# B&R Automation Studio project semesterProjekt_v002
Automation Studio 4.3.3.196

## Configuration Config1

### Task classes (Cpu.sw)
```
Cyclic#1 (cycle 1000 us, tolerance 1000 us):
  Program <- Program.prg
  reset <- reset.prg
Cyclic#4:
  emergencyS <- emergencyStop.prg
  TCP <- TCP.prg
VcDataObjects: Visu_R <- Visu_Resized.dob
Binaries: udbdef, TCData, vcrt, vcfntttf, Visu_R01, vcctext, Visu_R03, arial, vcmgr, vcpkat, vccovl, vccnum, vcpfar00, vcdsint, vcpfx20, vcpdvnc, vcshared, vcpdsw, vcfile, vcalarm, vccbtn, vcgclass, vcdsloc, arialbd, vcnet, vctcal, vcbclass, vccshape, Visu_R02, sysconf, Role, User, iomap, ashwd, asfw, arconfig, ashwac
Libraries: standard, astime, asieccon, fileio, dataobj, ashw, vcresman, AsMbTCP, runtime
```

### Hardware
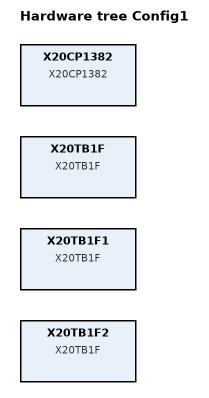
```
X20CP1382 : X20CP1382 v1.3.2.0  [X1 -> X1.SL; X2 -> X2.SL; X3 -> X3.SL]
  Module X1 (Type=X1, Virtual=true, Version=1.3.2.0)
    Connection (Connector=SS1, TargetModule=X20TB1F, TargetConnector=SS)
    Connection (Connector=SL, TargetModule=X20CP1382, TargetConnector=X1)
  Module X2 (Type=X2, Virtual=true, Version=1.3.2.0)
    Connection (Connector=SS1, TargetModule=X20TB1F1, TargetConnector=SS)
    Connection (Connector=SL, TargetModule=X20CP1382, TargetConnector=X2)
  Module X3 (Type=X3, Virtual=true, Version=1.3.2.0)
    Connection (Connector=SS1, TargetModule=X20TB1F2, TargetConnector=SS)
    Connection (Connector=SL, TargetModule=X20CP1382, TargetConnector=X3)
  Connector IF2:
    ActivateDevice = 1
    Mode = Manual
    InternetAddress = 192.168.0.103
    SubnetMask = 255.255.255.0
    Vnc1
    VncVcObjectName1 = Visu_R
    VncKeyMappingFile1 = VC\PS2-Keyboard.dis
    VncRefreshRate1 = 100
  ConfigurationID = semesterProjektTest_Config1
  VolatileGlobalPvSize = 655350
  SystemTick = 1000
  Cyclic1Duration = 1000
  Cyclic1Tolerance = 1000
X20TB1F : X20TB1F v1.0.0.0
X20TB1F1 : X20TB1F v1.0.0.0
X20TB1F2 : X20TB1F v1.0.0.0
```

## Logical view

Binary libraries used (declarations not repeated): operator, runtime, astime, AsIecCon, standard, AsMbTCP

### Global.var - Global variables
```iecst
VAR
	dirX : BOOL;
	dirY : BOOL;
	dirZ : BOOL;
	enabX : BOOL;
	enabY : BOOL;
	enabZ : BOOL;
	drawFunction : BOOL;
	input : ARRAY[0..1999999] OF UINT;
	posX : UDINT;
	posY : UDINT;
	posZ : UDINT;
	reset : BOOL;
	stepX : BOOL;
	stepY : BOOL;
	stepZ : BOOL;
	switch_X : BOOL;
	t : USINT;
	quit : BOOL;
	sharpen : UINT;
	status : USINT;
	testEnab : BOOL;
	z_move_down : BOOL;
	z_move_up : BOOL;
	y_move_right : BOOL;
	y_move_left : BOOL;
	x_move_right : BOOL;
	x_move_left : BOOL;
	sharpenderNeed : BOOL;
	switch_Z : BOOL;
	switch_Y : BOOL;
	percentage : REAL; (*%*)
	newLineX : UDINT;
	ValueZ : UINT;
	penLength : REAL;
	placeInString : UINT;
	placement : UINT;
	newLineHelper : UDINT;
END_VAR
```


### Program Logical/Program (IEC)

#### Main.st
```iecst
PROGRAM _INIT

	placeInString := 1;
	i := 0;
	sharpen := 1;
	activator := FALSE;
	testEnab:= FALSE;
	penLength := 0;
	sharpenderNeed:= 0;

END_PROGRAM

PROGRAM _CYCLIC
	ValueZ := REAL_TO_INT(penLength**1.5);

	IF (reset = FALSE AND testEnab = FALSE AND penLength > 5 ) THEN
//		percentage:= (UINT_TO_REAL(placeInString)/LEN(input))*100;

		IF (enabX = FALSE) THEN
			status:= 2;
		END_IF

		IF (i = 30) THEN
			placeInString := placeInString + 1;
			i := 0;
		END_IF
		placement := input[placeInString];

		// here the robot will move to the shapener, sharpen the pencil and move back to were it came from
		IF (sharpen = 1200 AND sharpenderNeed) THEN //!!!!!
			IF (posZ > 300 AND tempX > 0 AND activator = FALSE) THEN  // !!!!!!
				dirZ := TRUE;
				stepZ := NOT stepZ;
				IF (stepZ = FALSE) THEN
					posZ := posZ -1;
				END_IF

			ELSIF (tempX > 0 AND posZ = 300 AND activator = FALSE)THEN //!!!!!
				dirX := FALSE;
				stepX := NOT stepX;
				IF (stepX = FALSE) THEN
					tempX := tempX -1;
				END_IF

			ELSIF (tempX = 0 AND posZ < 1200 AND activator = FALSE) THEN //!!!!!
				dirZ := FALSE;
				stepZ := NOT stepZ;
				IF (stepZ = FALSE) THEN
					posZ := posZ +1;
				END_IF

			ELSIF (tempX = 0 AND posZ = 1200 AND activator = FALSE) THEN //!!!!!!
				timer.IN := TRUE;
				timer.PT := T#10000ms;
				IF timer.Q THEN
					activator := TRUE;
				END_IF

			ELSIF  (tempX = 0 AND posZ > 300 AND activator = TRUE) THEN//!!!!!
				dirZ := TRUE;
				stepZ := NOT stepZ;
				IF (stepZ = FALSE) THEN
					posZ := posZ - 1;
				END_IF

			ELSIF (tempX < posX  AND posZ = 300 AND activator = TRUE) THEN //!!!!!
				dirX := TRUE;
				stepX := NOT stepX;
				IF (stepX = FALSE) THEN
					tempX := tempX +1;
				END_IF

			ELSIF (tempX = posX  AND posZ = 300 AND activator = TRUE) THEN //!!!!!!
				sharpen := 0;
				activator := FALSE;

			END_IF

		ELSE
			// here the robot will draw
			IF (placement = 21041 AND i < 30) THEN
				IF (posZ < (3200-ValueZ)) THEN  // !!!!!!
						dirZ := TRUE;
						stepZ := NOT stepZ;
						IF (stepZ = FALSE) THEN
							posZ := posZ +1;
						END_IF

					ELSE
						dirX := TRUE;
						stepX := NOT stepX;
						IF (stepX = FALSE) THEN
							posX := posX + 1;
							newLineX := newLineX +1;
							sharpen := sharpen + 1;
							tempX := posX;
						END_IF
						i := i + 1;
					END_IF

			//dont draw
			ELSIF placement = 21040 AND i < 30) THEN

				IF (posZ > (2900-ValueZ)) THEN  // !!!!!!
						dirZ := FALSE;
						stepZ := NOT stepZ;
						IF (stepZ = FALSE) THEN
							posZ := posZ -1;
						END_IF

					ELSE
						dirX := TRUE;
						stepX := NOT stepX;
						IF (stepX = FALSE) THEN
							posX := posX +1;
							newLineX := newLineX +1;
						END_IF
						i := i + 1;

				ELSIF (i = 3) THEN
					placeInString := placeInString + 1;
					i := 0;

//				ELSE
//					placeInString := placeInString + 1;

				END_IF

//			ELSIF (placement = '1' OR placement = '0') THEN
//				placeInString := placeInString + 1;

			ELSIF (placement = 20016 OR placement = 20017) THEN
				IF (posZ > (2900-ValueZ) )THEN  // !!!!!!
					dirZ := FALSE;
					stepZ := NOT stepZ;
					IF (stepZ = FALSE) THEN
						posZ := posZ -1;
					END_IF
				ELSIF (posZ = (2900-ValueZ)) AND (newLineX >= (newLineHelper)) THEN//!!!!
					dirX := FALSE;
					stepX := NOT stepX;
					IF (stepX = FALSE) THEN
						posX := posX - 1;
						newLineX := newLineX -1;
					END_IF

				ELSIF ((posZ = (2900-ValueZ)) AND (newLineX <= newLineHelper) AND (i <= 30)(* OR ( posZ = 0)*)) THEN
					dirY := TRUE;
					stepY := NOT stepY;
					IF (stepY = FALSE) THEN
						posX := posX - 1;
						newLineX := newLineX -1;

					END_IF

					i := i +1;
				END_IF

				IF i = 20 THEN
					newLineHelper := newLineHelper - 12 ;

				END_IF

			ELSIF (placement = 20785 or placement = 20784) THEN

				quit := TRUE;
			END_IF

		END_IF

	END_IF
END_PROGRAM

PROGRAM _EXIT
	(* Insert code here *)

END_PROGRAM
```

### Program Logical/reset (IEC)

#### Main.st
```iecst
PROGRAM _INIT
	reset := TRUE;//!!!!!!!!
	resetX := 0;
	resetY := 0;
	resetZ := 0;

	quit := FALSE;
	status := 1;
	testEnab := TRUE;//!!!!!!
	posX := 0;
	posY := 0;
	posZ := 0;

END_PROGRAM

PROGRAM _CYCLIC

// resets x-, y- and z-axis.
	IF (reset = TRUE AND testEnab = FALSE) THEN
		IF switch_X = TRUE AND resetX = 0  THEN
			enabX:= FALSE;
			dirX:= FALSE;
			stepX := NOT stepX;
		ELSIF switch_X = FALSE THEN
			resetX := 1;
			dirX:= TRUE;
			stepX := NOT stepX;
		END_IF

		IF switch_Y = TRUE AND resetY = 0 THEN
			enabY:= FALSE;
			dirY:= FALSE;
			stepY := NOT stepY;
		ELSIF switch_Y = FALSE THEN
			resetY := 1;
			dirY:= TRUE;
			stepY := NOT stepY;
		END_IF

		IF switch_Z = TRUE AND resetZ = 0 THEN
			enabZ:= FALSE;
			dirZ:= FALSE;
			stepZ := NOT stepZ;
		ELSIF switch_Z = FALSE THEN
			resetZ := 1;
			dirZ:= TRUE;
			stepZ := NOT stepZ;
		END_IF
// sets the position of the variables posX, posY and posZ
		timer.IN := TRUE;
		timer.PT := T#100ms;
		IF timer.Q THEN
			IF resetX = 1 AND resetY = 1 AND resetZ = 1 THEN
				posX := 0;
				posY := 0;
				posZ := 0;
				resetX := 2;
			END_IF
			timer.IN := FALSE;
		END_IF

	// if start-button pressed, then go to start position
		IF quit = FALSE AND resetX = 2 THEN
			IF posX < 1900 THEN
				dirX := TRUE;
				stepX := NOT stepX;
				IF (stepX = FALSE) THEN
					posX := posX +1;
				END_IF
			ELSE
				reset:= FALSE;
				resetX := 0;
				resetY := 0;
				resetZ := 0;
				newLineX :=  2294967295;
				newLineHelper := 2294967295;
			END_IF
		END_IF
	END_IF

	// move x-axis left
	IF (x_move_left AND testEnab) THEN
		stepX := NOT stepX;
		dirX := TRUE;
		IF stepX = FALSE THEN
			posX := posX +1;
		END_IF
	END_IF

	// move x-axis right
	IF (x_move_right AND testEnab) THEN
		stepX := NOT stepX;
		dirX := FALSE;
		IF stepX = FALSE THEN
			posX := posX -1;
		END_IF
	END_IF

	// move y-axis left
	IF (y_move_left AND testEnab) THEN
		stepY := NOT stepY;
		dirY := TRUE;
		IF stepY = FALSE THEN
			posY := posY +1;
		END_IF
	END_IF

	// move y-axis right
	IF (y_move_right AND testEnab) THEN
		stepY := NOT stepY;
		dirY := FALSE;
		IF stepY = FALSE THEN
			posY := posY -1;
		END_IF
	END_IF

	// move z-axis up
	IF (z_move_up AND testEnab) THEN
		stepZ := NOT stepZ;
		dirZ := FALSE;
		IF stepZ = FALSE THEN
			posZ := posZ -1;
		END_IF
	END_IF

	// move z-axis down
	IF (z_move_down AND testEnab) THEN
		stepZ := NOT stepZ;
		dirZ := TRUE;
		IF stepZ = FALSE THEN
			posZ := posZ +1;
		END_IF
	END_IF

	timer();
END_PROGRAM

PROGRAM _EXIT
	(* Insert code here *)

END_PROGRAM
```

### Program Logical/emergencyStop (IEC)

#### Variables.var
```iecst
VAR
	emergencyStop : BOOL;
	reset_quit : BOOL;
END_VAR
```

#### Main.st
```iecst
PROGRAM _INIT
	(* Insert code here *)
	reset_quit := FALSE;
	emergencyStop := FALSE;

END_PROGRAM

PROGRAM _CYCLIC
	IF (emergencyStop) THEN
		enabX := TRUE;
		enabY := TRUE;
		enabZ := TRUE;
		status := 0;

	END_IF

	IF (reset_quit) THEN
		reset := TRUE;
		quit := TRUE;
		status := 1;
		reset_quit := FALSE;
		placeInString :=1;

	END_IF

END_PROGRAM

PROGRAM _EXIT
	(* Insert code here *)

END_PROGRAM
```

- Visualisation Logical/Visu_Resized (not shown)

### Program Logical/TCP (IEC)

#### Main.st
```iecst
PROGRAM _INIT
	state := 1;

END_PROGRAM

PROGRAM _CYCLIC
	CASE state OF
		1:
			tcp1.enable := TRUE;
			tcp1.port := 12345;
			tcp1.options := tcpOPT_REUSEADDR;
			tcp1();
			IF tcp1.status = 0 THEN
				state := 10;
			END_IF

		10:
			tcp2.enable := TRUE;
			tcp2.ident := tcp1.ident;
			tcp2();
			IF tcp2.status = 0 THEN
				state := 20;
			END_IF

		20:
			tcp3.enable := TRUE;
			tcp3.ident := tcp2.identclnt;
			tcp3.pData := ADR(reciveData);
			tcp3.datamax := SIZEOF (reciveData);
			tcp3();
			IF tcp3.status = 0 THEN
				sendData := reciveData;
				//				FOR i := 0 TO i = 2000 BY i + 1 DO
				//					test.IN := reciveData[i];
				//					input := CONCAT(input, test.Q);
				//				END_FOR
				state := 30;

			END_IF

		30:
			tcp4.enable := TRUE;
			tcp4.ident := tcp2.identclnt;
			tcp4.pData := ADR(sendData);
			tcp4.datalen := brsstrlen(ADR(sendData));
			tcp4();
			IF tcp4.status = 0 THEN
				state := 40;
			END_IF

		40:
			tcp5.enable := TRUE;
			tcp5.ident := tcp2.identclnt;
			tcp5();
			IF tcp5.status = 0 THEN
				tcp2.enable := FALSE;
				state := 10;

				//				FOR i := 0 TO i < 200 BY i + 1 DO
				//					reciveData[i] := 0;
				//				END_FOR
			END_IF
	END_CASE
	test();
END_PROGRAM

PROGRAM _EXIT
	tcp5.enable := TRUE;
	tcp5.ident := tcp2.identclnt;
	tcp5();

	tcp5.enable := TRUE;
	tcp5.ident := tcp1.ident;
	tcp5();
```

Listed in the project but not available here: Logical/Global.typ
